// TIA Portal V17 export
// export: Created 2026-04-13T11:12:41.3455714Z, ExportSetting WithDefaults, DisplayName Totally Integrated Automation Portal, DisplayVersion V17 Update 4, DisplayName TIA Portal Openness, DisplayVersion V17 Update 4, DisplayName TIA Portal Version Control Interface, DisplayVersion V17, DisplayName SINAMICS Startdrive Advanced, DisplayVersion V17, DisplayName SINAMICS Startdrive G130, G150, S120, S150, SINAMICS MV, S210, DisplayVersion V17, DisplayName SINAMICS Startdrive G110M, G120, G120C, G120D, G120P, G115D, DisplayVersion V17, DisplayName STEP 7 Professional, DisplayVersion V17 Update 4, DisplayName STEP 7 Safety, DisplayVersion V17, DisplayName WinCC Professional, DisplayVersion V17 Update 4
FUNCTION_BLOCK "A2-数据转换ITR"   // FB56, SCL
{ S7_Optimized_Access := 'TRUE' }
VERSION : 0.1
// stored: AutoNumber true, IsIECCheckEnabled false, IsRetainMemResEnabled false, MemoryReserve 100, SetENOAutomatically false, UDAEnableTagReadback false
   VAR_INPUT
      I_ChValue : Int;   // 通道值输入
      I_Max : Int := 27648;
      I_Min : Int := 0;
      R_Max : Real;   // 仪表物理最大值(设置值)
      R_Min : Real;   // 仪表物理最小值(设置值)
      R_Edit : Real;   // 数值修订
      R_HHAlarm_Set : Real;   // 超高报警限值(设置值)
      R_HAlarm_Set : Real;   // 高报警限值(设置值)
      R_LAlarm_Set : Real;   // 低报警限值(设置值)
      R_LLAlarm_Set : Real;   // 超低报警限值(设置值)
   END_VAR
   VAR_OUTPUT
      R_Meter_Value : Real;   // 仪表实时值(输出值)
      b_HH_Alarm : Bool;   // 超高报警
      b_H_Alarm : Bool;   // 高报警
      b_L_Alarm : Bool;   // 低报警
      b_LL_Alarm : Bool;   // 超低报警
      Status : Int;   // 状态值
   END_VAR
   VAR
      input : Int;
   END_VAR
BEGIN
   (*
       数据转换AI通道值转换成仪表值
       OUT = [((FLOAT (IN) – K1)/(K2–K1)) * (HI_LIM–LO_LIM)] + LO_LIM
    *)
   (*传感器状态:0,正常;1,溢出;2:故障.*)
   IF  #I_ChValue =32767 OR #I_ChValue =-32768 THEN    //仪表故障
       #input := 0;
       #Status := 2;
   ELSIF
       #I_ChValue > 28000 AND #I_ChValue <32767 THEN   //通道溢出
       #input := 27648;
       #Status := 1;
   ELSIF #I_ChValue < -100 AND #I_ChValue >-32768 THEN   //通道溢出
       #input := 0;
       #Status := 1;
   ELSE
       #input := #I_ChValue;  //仪表正常
       #Status := 0;
   END_IF;

   #R_Meter_Value := ((INT_TO_REAL(#input)-#I_Min) / (#I_Max-#I_Min)) * (#R_Max - #R_Min) + #R_Min + #R_Edit; //仪表值计算

   IF  #R_Meter_Value >= #R_HHAlarm_Set THEN      //超高报警
       #b_HH_Alarm := 1;
   ELSE
       #b_HH_Alarm := 0;
   END_IF;

   IF #R_Meter_Value >= #R_HAlarm_Set THEN      //高报警
       #b_H_Alarm := 1;
   ELSE
       #b_H_Alarm := 0;
   END_IF;

   IF #R_Meter_Value <= #R_LLAlarm_Set THEN      //超低报警
       #b_LL_Alarm := 1;
   ELSE
       #b_LL_Alarm := 0;
   END_IF;

   IF #R_Meter_Value <= #R_LAlarm_Set THEN      //低报警
       #b_L_Alarm := 1;
   ELSE
       #b_L_Alarm := 0;
   END_IF;
END_FUNCTION_BLOCK
